FUNCTION_BLOCK XtsMoverAxis EXTENDS CyclicBase IMPLEMENTS ITF_XtsMoverAxis
VAR
	MyAxisRef : AXIS_REF;
	_MyAxisStatus : ST_AxisStatus;
	_MyNCData : NCTOPLC_AXIS_REF;
	MoverPowerCommand : AxisPower(MyAxisRef);
	MoverMoveCommand : MoveModuloMoverToPosition(MyAxisRef) := (Gap := 100.0);
	MoverHaltCommand : HaltMover(MyAxisRef);
	MoverResetCommand : AxesReset(MyAxisRef);
	MoverActivateTrackCommand : ActivateTrackForMover(MyAxisRef);
	axesGear	: GearInCA(MyAxisRef);
	_ipTcIoXtsMover	: I_TcIoXtsXpuMover;
	_ActiveTrackLength : MC_LREAL;
	TrackChangeTrigger : R_TRIG;
	_MoverAbsMoveOptions : ST_MoveAbsoluteCAOptions;
	_stTmsActPositions			: ST_PositionInfo;
	_CurrentTrack : I_XtsTrack;
	_MyCAGroup : ICollisionGroup;
	_ForwardOnly : BOOL := TRUE;
END_VAR
VAR CONSTANT
	_MaxMoverVelocity : MC_LREAL := 4000.0;
END_VAR

PROPERTY PUBLIC Acceleration : MC_LREAL
GET
Acceleration := MoverMoveCommand.Acceleration;
END_GET
SET
MoverMoveCommand.Acceleration := Acceleration;
END_SET
END_PROPERTY

METHOD ActivateTrack : HRESULT
VAR_INPUT
	NewTrack : OTCID;
	Track : I_XtsTrack;
END_VAR
IF NOT MoverActivateTrackCommand.Busy AND THIS^.isMoverStationary() AND NewTrack <> 0  THEN
	IF MoverActivateTrackCommand.Execute(Track := Track.MyOTCID) THEN
		_CurrentTrack := Track;
		_ActiveTrackLength := Track.TrackLength;
		ActivateTrack := 1;
	ELSE
		ActivateTrack := -1;
	END_IF
ELSE
	ActivateTrack := -1;
END_IF
END_METHOD

METHOD ActivateZeroReferenceSystem : HRESULT
VAR_INPUT
	NewTrack : OTCID;
END_VAR
IF NOT MoverActivateTrackCommand.Busy AND THIS^.isMoverStationary() THEN // AND NewTrack <> 0  THEN
	IF MoverActivateTrackCommand.Execute(Track := NewTrack) THEN
		_CurrentTrack := 0;
		ActivateZeroReferenceSystem := 1;
	ELSE
		ActivateZeroReferenceSystem := -1;
	END_IF
ELSE
	ActivateZeroReferenceSystem := -1;
END_IF
END_METHOD

PROPERTY AxisRef : Reference to Axis_ref
GET
AxisRef REF= MyAxisRef;
END_GET
END_PROPERTY

METHOD PUBLIC  Cycle : HRESULT
VAR_INPUT
END_VAR
IF isMoverDetected() THEN
	MoverPowerCommand.Cycle();
	MoverMoveCommand.Cycle();
	MoverHaltCommand.Cycle();
	MoverResetCommand.Cycle();
	MoverActivateTrackCommand.Cycle();
	axesGear.Cycle();
	TrackChangeTrigger(CLK := MoverActivateTrackCommand.Done);
	IF TrackChangeTrigger.Q THEN
		_MoverAbsMoveOptions.PositionReferenceSystem :=  MoverActivateTrackCommand.NewTrackId;
		_MoverAbsMoveOptions.DynamicsReferenceSystem := MoverActivateTrackCommand.NewTrackId;
		MoverMoveCommand.Options := _MoverAbsMoveOptions;	
	END_IF
	IF _ipTcIoXtsMover <> 0 THEN
		_stTmsActPositions := _ipTcIoXtsMover.GetPositionInfo();
	END_IF
	Cycle := 1;
ELSE
	Cycle := -1;
END_IF
MyAxisRef.ReadStatus();
_MyNCData := MyAxisRef.NcToPlc;
_MyAxisStatus := MyAxisRef.Status;
END_METHOD

PROPERTY PUBLIC Deceleration : MC_LREAL
GET
Deceleration := MoverMoveCommand.Deceleration;
END_GET
SET
MoverMoveCommand.Deceleration := Deceleration;
MoverHaltCommand.Deceleration := Deceleration;
END_SET
END_PROPERTY

METHOD PUBLIC DisableMover : HRESULT
VAR_INPUT
END_VAR
IF THIS^.isMoverEnabled() AND NOT MoverPowerCommand.Busy THEN
	MoverPowerCommand.Disable();
	DisableMover := 1;
ELSE
	DisableMover := -1;
END_IF
END_METHOD

METHOD PUBLIC EnableMover : HRESULT
VAR_INPUT
END_VAR
IF (NOT MoverPowerCommand.Busy) AND NOT THIS^.isMoverEnabled() THEN // AND _CurrentTrack <> 0 THEN
	MoverPowerCommand.Enable();
	EnableMover := 1;
ELSE
	EnableMover := -1;
END_IF
END_METHOD

PROPERTY PUBLIC Gap : MC_LREAL
GET
Gap := MoverMoveCommand.Gap;
END_GET
SET
IF Gap >= 50.0 THEN
	MoverMoveCommand.Gap := Gap;
	MoverHaltCommand.Gap := Gap;
ELSE
	Gap := 100.0;
END_IF
END_SET
END_PROPERTY

METHOD PUBLIC Gear : HRESULT
VAR_INPUT
	MasterPosition : MC_LREAL;
	SlavePosition : MC_LREAL;
END_VAR
IF NOT axesGear.Busy AND __ISVALIDREF(axesGear.MyGearMaster) AND MasterPosition <= _ActiveTrackLength AND SlavePosition <= _ActiveTrackLength THEN
	IF axesGear.Sync(MasterPosition := MasterPosition, SlavePosition := SlavePosition) THEN
		Gear := 1;
	ELSE
		Gear := -1;
	END_IF
ELSE
	Gear := -1;
END_IF
END_METHOD

METHOD GetMoverCtrlOTCID : XtsMoverControllerOTCID
VAR_INPUT
END_VAR
GetMoverCtrlOTCID := _ipTcIoXtsMover.P_MoverControllerOid;
END_METHOD

METHOD GetMoverOTCID : OTCID
VAR_INPUT
END_VAR
//GetMoverCtrlOTCID := _ipTcIoXtsMover.P_AxisOid;
END_METHOD

METHOD PUBLIC HaltAxis : HRESULT
VAR_INPUT
END_VAR
IF NOT MoverHaltCommand.Busy THEN// AND NOT THIS^.isMoverStationary() THEN
	IF MoverHaltCommand.Execute() THEN
		HaltAxis := 1;
	ELSE
		HaltAxis := -1;
	END_IF
ELSE
	HaltAxis := -1;
END_IF
END_METHOD

PROPERTY PUBLIC IdentInGroup : IDENT_IN_GROUP_REF
GET
IdentInGroup := UDINT_TO_IDENTINGROUP(id := _MyNCData.AxisId);
END_GET
END_PROPERTY

METHOD inGear : BOOL
VAR_INPUT
END_VAR
inGear := axesGear.GearInPosCA.InSync;
END_METHOD

METHOD IsActive : BOOL
VAR_INPUT
END_VAR
IsActive := _ipTcIoXtsMover.GetIsActive();
END_METHOD

METHOD PUBLIC isMoverAtPosition : BOOL
VAR_INPUT
	Position : MC_LREAL;
END_VAR
IF Position > 1 THEN
	IF _stTmsActPositions.fTrackPosition < position + 1 AND _stTmsActPositions.fTrackPosition > position - 1 THEN
		isMoverAtPosition := TRUE;
	ELSE
		isMoverAtPosition := FALSE;
	END_IF  
ELSE
	IF _stTmsActPositions.fTrackPosition < position + 1 AND _stTmsActPositions.fTrackPosition > 0.0  
		OR _stTmsActPositions.fTrackPosition < _CurrentTrack.TrackLength AND _stTmsActPositions.fTrackPosition > _CurrentTrack.TrackLength - 1 THEN
		isMoverAtPosition := TRUE;
	ELSE
		isMoverAtPosition := FALSE;
	END_IF
END_IF
END_METHOD

METHOD PUBLIC isMoverDetected : BOOL
VAR_INPUT
END_VAR
isMoverDetected := _MyNCData.AxisId <> 0;
END_METHOD

METHOD PUBLIC isMoverEnabled : BOOL
VAR_INPUT
END_VAR
isMoverEnabled :=  NOT _MyAxisStatus.Disabled;
END_METHOD

METHOD PUBLIC isMoverStationary : BOOL
VAR_INPUT
END_VAR
isMoverStationary := _MyAxisStatus.NotMoving;
END_METHOD

PROPERTY PUBLIC Jerk : MC_LREAL
GET
Jerk := MoverMoveCommand.Jerk;
END_GET
SET
MoverMoveCommand.Jerk := Jerk;
MoverHaltCommand.Jerk := Jerk;
END_SET
END_PROPERTY

PROPERTY PUBLIC MoverErrorID : DWORD
GET
MoverErrorID := _MyAxisStatus.ErrorID;
END_GET
END_PROPERTY

PROPERTY PUBLIC MoversActiveTrack : OTCID
GET
MoversActiveTrack := _ipTcIoXtsMover.GetActiveTrackObjectId();
END_GET
END_PROPERTY

PROPERTY PUBLIC MoverXtsIoEnvInterface : I_TcIoXtsXpuMover
GET
MoverXtsIoEnvInterface := _ipTcIoXtsMover;
END_GET
SET
_ipTcIoXtsMover := MoverXtsIoEnvInterface;
END_SET
END_PROPERTY

METHOD PUBLIC MoveTo : HRESULT
VAR_INPUT
	RequiredPosition : MC_LREAL;
	MoveVelocity : MC_LREAL;
	NonModuloMove : BOOL;
END_VAR
IF NOT MoverMoveCommand.Busy AND MoveVelocity < _MaxMoverVelocity AND MoveVelocity > 0.0 AND Gap >= 50.0 THEN
	IF NonModuloMove THEN
		IF THIS^.MoverMoveCommand.MoveTo(Position := RequiredPosition, 
										Velocity := MoveVelocity, 
										Direction := Tc3_Mc3Definitions.MC_DIRECTION.mcDirectionNonModulo, 
										Turns := 0) THEN
										
			MoveTo := 1;
		END_IF
	ELSE
		IF _ForwardOnly THEN
			THIS^.MoverMoveCommand.MoveTo(Position := RequiredPosition, 
										Velocity := MoveVelocity, 
										Direction := Tc3_Mc3Definitions.MC_DIRECTION.mcDirectionPositive, 
										Turns := 0);
			MoveTo := 1;
		ELSE
			IF RequiredPosition > MyAxisRef.NcToPlc.ModuloActPos THEN
				IF THIS^.MoverMoveCommand.MoveTo(Position := RequiredPosition, 
											Velocity := MoveVelocity, 
											Direction := Tc3_Mc3Definitions.MC_DIRECTION.mcDirectionPositive, 
											Turns := 0) THEN
											
					MoveTo := 1;
				END_IF
			ELSE
				IF THIS^.MoverMoveCommand.MoveTo(Position := RequiredPosition, 
											Velocity := MoveVelocity, 
											Direction := Tc3_Mc3Definitions.MC_DIRECTION.mcDirectionNegative, 
											Turns := 0) THEN
											
					MoveTo := 1;
				END_IF	
			END_IF
		END_IF
	END_IF
ELSE
	MoveTo := -1;
END_IF
END_METHOD

PROPERTY MyCAGroup : ICollisionGroup
GET
MyCAGroup := _MyCAGroup;
END_GET
SET
_MyCAGroup := MyCAGroup;
END_SET
END_PROPERTY

PROPERTY MyMasterRef : REFERENCE TO AXIS_REF
GET
MyMasterRef REF= axesGear.MyGearMaster;
END_GET
SET
axesGear.MyGearMaster REF= MyMasterRef;
END_SET
END_PROPERTY

PROPERTY PositiveDirectionOnly : BOOL
GET
PositiveDirectionOnly := _ForwardOnly;
END_GET
SET
_ForwardOnly := PositiveDirectionOnly;
END_SET
END_PROPERTY

METHOD PUBLIC ResetAxis : HRESULT
VAR_INPUT
END_VAR
IF NOT MoverResetCommand.Busy AND _MyAxisStatus.Error THEN
	IF MoverResetCommand.Execute() = S_OK THEN
		ResetAxis := 1;
	ELSE
		ResetAxis := -1;
	END_IF
ELSE
	ResetAxis := -1;
END_IF
END_METHOD

METHOD SetForceCouple : HRESULT
VAR_INPUT
	XtsMoverCtrlOTCID : Tc3_XTS_Utility.XtsMoverControllerOTCID;
END_VAR
_ipTcIoXtsMover.MoverController.SetForceCouple(nForceCouple := XtsMoverCtrlOTCID);
END_METHOD

METHOD SwapMover : HRESULT
VAR_INPUT
    MoverToSwapWith : MoverOTCID;
END_VAR
_ipTcIoXtsMover.swapmover(nSwapMoverObjectId := MoverToSwapWith);
END_METHOD

METHOD TriggerMoverArrive : BOOL
VAR_INPUT
END_VAR
_ipTcIoXtsMover.TriggerArrive();
END_METHOD

METHOD TriggerMoverLeave : BOOL
VAR_INPUT
END_VAR
TriggerMoverLeave := _ipTcIoXtsMover.TriggerLeave();
END_METHOD

END_FUNCTION_BLOCK

(* stored: Version 1.1.0.1
   POU XtsMoverAxis: Id {f9a43ed2-0578-4aed-857c-1a3adef0c7f6}, SpecialFunc None
   Folder Administration: Id {660864df-8996-42d7-8e95-bfca1c90696e}
   Folder Commands: Id {db0a893b-cc1a-482e-a432-7e9d568c5112}
   Folder Dynamics: Id {6b49cc7a-c913-475a-9f9a-db91d65d07e1}
   Folder ICyclic: Id {895ad701-1670-4c6d-921e-cd7ccab0c12a}
   Folder Status: Id {b27ba391-8a3b-4e51-ae24-bae43a7b6e5f}
   Property Acceleration: Id {5cd04126-8ceb-4f9d-a4c5-c87e7e11d0e6}
   Get Get: Id {89c9e6d0-5dfa-4531-97de-32e16eb2e196}
   Set Set: Id {95cc2e62-d911-4757-83d0-b9b38a36fdde}
   Method ActivateTrack: Id {f7604675-5338-4e11-9132-b17d5df72cc8}
   Method ActivateZeroReferenceSystem: Id {f593e12a-c440-483d-8309-49c5dc48d5f1}
   Property AxisRef: Id {a7d5ea1d-51bb-4c87-90b3-db66fd196d20}
   Get Get: Id {8c3b00e4-86fb-42e3-b0e0-5789e5045419}
   Method Cycle: Id {b5956233-12ba-4cb8-805f-5693aec42bed}
   Property Deceleration: Id {3def2bbc-f7ec-4120-acb9-2ff2a2789bd5}
   Get Get: Id {e6097884-8279-4e20-92f9-6fb8b5120af4}
   Set Set: Id {dbf3cf03-c8db-40c9-ab3e-669bb5cdced1}
   Method DisableMover: Id {a82f95fa-77b4-4c5e-ae67-686dbd3b2d8d}
   Method EnableMover: Id {d130fe63-f34a-4455-8bb8-4dfcc482e573}
   Property Gap: Id {dd72da9d-fc94-421a-8ee7-a84a721dd20c}
   Get Get: Id {5c8fd02d-70e7-4f46-b386-6000a46a3487}
   Set Set: Id {280f9258-e1cd-43be-bf57-16929cbbc8d6}
   Method Gear: Id {b0aa32af-e1ad-43df-b90e-7e7d830bc963}
   Method GetMoverCtrlOTCID: Id {6852d0c0-13fb-4a6d-9e8b-5d538e770d2f}
   Method GetMoverOTCID: Id {0ee3ade7-076c-46ec-8833-0ad2fc45f400}
   Method HaltAxis: Id {b177db81-8e99-498a-a7a2-cd0938dd7a2c}
   Property IdentInGroup: Id {4d5563a0-634a-4074-a0e4-612875dd790c}
   Get Get: Id {6419a53d-e416-464a-881c-e300db0a9add}
   Method inGear: Id {0809336a-3200-4d64-8806-8b040d87d191}
   Method IsActive: Id {4093fe18-48a9-45f2-9701-210b5183f8f4}
   Method isMoverAtPosition: Id {f1a74560-cd92-4fa6-83a2-3bacea608337}
   Method isMoverDetected: Id {c1a5811f-71c0-458a-bf03-7bfa946db86b}
   Method isMoverEnabled: Id {7f5530a3-9bf6-4669-8c7b-76814da68801}
   Method isMoverStationary: Id {64b09804-b6c0-46e5-9180-be650a88cf77}
   Property Jerk: Id {fbc5f504-aa6b-48f8-8a62-bbde3b74b20e}
   Get Get: Id {98c0c9db-aae6-4788-a223-2bf5fa007418}
   Set Set: Id {6a6a16a3-4f19-4f4d-bd8d-8441ae3b5cf2}
   Property MoverErrorID: Id {9a24b894-1b02-4293-95b1-831b38fd5fad}
   Get Get: Id {01f9b7c9-0e41-48f0-a5f9-8a7a495677b0}
   Property MoversActiveTrack: Id {15471ba0-8341-48c7-a2d0-01ca6286078a}
   Get Get: Id {2721855b-e1d8-4f74-a352-28794ee4ae69}
   Property MoverXtsIoEnvInterface: Id {6aaf98f4-e1bc-4f35-afbe-48664404e767}
   Get Get: Id {5b75808a-7c24-4c09-8809-4a555d5acdb1}
   Set Set: Id {57119448-dfbf-405e-ade1-72aad5224720}
   Method MoveTo: Id {ea6488b0-fefd-4f9f-a3b2-cfd8c6f64d05}
   Property MyCAGroup: Id {ef4ebc28-e3bd-4e4a-8472-4104ad14ebae}
   Get Get: Id {d4b3e253-6981-43ac-859c-776f6b4fec7d}
   Set Set: Id {54c77228-8f9c-4310-9bfc-ef466b7143ba}
   Property MyMasterRef: Id {9a3e9617-3bee-43bf-8371-dedd27acecb0}
   Get Get: Id {d8c8a090-d5eb-4847-8f12-c276f8e68cfb}
   Set Set: Id {f5a13744-c943-4208-a476-90f7059f62be}
   Property PositiveDirectionOnly: Id {993fe16b-05a5-4eca-a38c-6463f3e7295c}
   Get Get: Id {581a1e54-141a-440c-9d85-39be9d6e8e36}
   Set Set: Id {aede2ad8-809d-4697-b667-b49152253954}
   Method ResetAxis: Id {e9d8249c-2f88-4980-a483-ceda82c7ab80}
   Method SetForceCouple: Id {655fe1cd-78c7-4097-b5c7-b05e68cd5f7e}
   Method SwapMover: Id {075d081f-a4ad-470f-95aa-ced1f28cc5a8}
   Method TriggerMoverArrive: Id {9bb7f072-ab21-4ec2-9434-ad1366cf5fb7}
   Method TriggerMoverLeave: Id {074e60e5-1df3-46d8-92fd-930fc05fcb13} *)
